(* IEC 61131-3 sources: paho.mqtt.c-ar/Samples/IotMqttSamples/SampleTasks/IotMqttConfig, 2 files *)

(* ---- Main.st ---- *)
PROGRAM _INIT
    IotMqttConfigParams.UseFile               := TRUE;
    IotMqttConfigParams.LogFileDevice	      := 'USER';
    IotMqttConfigParams.LogFileName		      := 'IotMqttLog';
    IotMqttConfigParams.AppendTimestamp	      := FALSE;
    IotMqttConfigParams.OverwritteLogs	      := TRUE;
    IotMqttConfigParams.LogLevel		      := IOTMQTT_LOG_LEVEL_ERROR;
    IotMqttConfig(ADR(IotMqttConfigParams));
END_PROGRAM

(* ---- Variables.var ---- *)
VAR
	IotMqttConfigParams : IotMqttConfigParametersType;
END_VAR
